Staubli VAL3: mcp.pgx

program mcp()
begin

  title("Pirámide")

  userPage()

  while !bFin
    // Se borra la pantalla
    cls()

    // Se muestra informacion en la pantalla
    gotoxy(2,3)
    put("Total  = "+toString("4",nPlantas))
    gotoxy(2,4)
    put("Actual = "+toString("4",nNivel))
    gotoxy(7,7)
    put(sMensaje)

    // Se muestran las etiquetas de las teclas de funcion
    gotoxy(0,13)
    put("Pir.")
    gotoxy(10,13)
    put("Edit")
    gotoxy(35,13)
    put("Fin")

    // Se procesa la tecla pulsada
    nTecla=getKey()
    switch nTecla
      // Enter - Orden de continuar
      case 270
        bPiezaPreparada=true
      break
      // F1 - Orden de construir piramide
      case 271
        bStartPiramide=true
      break
      // F3 - Orden de editar el numero de plantas a construir
      case 273
        //Obtener n
        gotoxy(1,1)
        put("Introduzca nº plantas")
        gotoxy(23,1)
        get(nPlantas)
      break
      // F8 - Orden de salir de la aplicacion
      case 278
        bTermina=true
      break
    endSwitch
    // Se da paso a la siguiente tarea y se estabiliza la pantalla
    delay(0.1)
  endWhile
  bFin=false
  // Se muestra un mensaje de despedida
  cls()
  gotoxy(12,7)
  put("Programa terminado")

end
